// Mitsubishi GX Works2 project: finalfinal[1]   PLC: FX3G

// global labels: Global1
VAR_GLOBAL
  startDaySwitch AT X007 : BOOL;
  petelValue AT D1111 : REAL;
  petelTank AT D1101 : REAL;
  lemonValue AT D1114 : REAL;
  lemonTank AT D1103 : REAL;
  GummyBear AT D1118 : REAL;
  GummyBearTank AT D1120 : REAL;
  stabillizerValue AT D1106 : REAL;
  stabillizerTank AT D1127 : REAL;
  totalPackages AT D1108 : REAL;
  finished_timer AT TS5 : BOOL;
  GummyGumPackages AT D1108 : INT;
END_VAR
VAR_GLOBAL CONSTANT
  zeroPackages : REAL;
  amountOfPetelForOnePackage : REAL := 280;
  amountOfLemonForOnePackage : REAL := 455;
  amountOfStabillizerForOnePackage : REAL := 105;
  amountOfGummyBearForOnePackage : REAL := 28;
END_VAR
VAR_GLOBAL
  notEnoughForRegularGummyGam AT M23 : BOOL;
  notEnoughForPinukGummyGam AT M24 : BOOL;
END_VAR
VAR_GLOBAL CONSTANT
  amountOfPetelForPinukPack : REAL := 385;
  amountOfLemonForPinukPack : REAL := 665;
  amountOfStabillizerForPinukPack : REAL := 210;
  amountOfGummyBearForPinukPack : REAL := 70;
END_VAR
VAR_GLOBAL
  endDay AT M25 : BOOL;
  dayOn AT Y007 : BOOL;
  Sample AT X001 : BOOL;
  analogInput1 AT D8280 : INT;
  save AT D8000 : INT;
  saveAnalogInput AT D8000 : INT;
END_VAR
VAR_GLOBAL CONSTANT
  normalizeAnalog : REAL := 400;
END_VAR
VAR_GLOBAL
  gumygamType AT D1333 : REAL;
  chekType AT M116 : BOOL;
END_VAR
VAR_GLOBAL CONSTANT
  pinukThreshold : REAL := 5.0;
END_VAR
VAR_GLOBAL
  notEnoughMaterials AT M26 : BOOL;
  emergency AT X005 : BOOL;
END_VAR
VAR_GLOBAL CONSTANT
  amountOfPetel : REAL := 280;
  amountOfPetelP : REAL := 385;
  amountOfLemon : REAL := 665;
  amountOfLemonP : REAL := 665;
  amountOfStabillizerP : REAL := 210;
  amountOfPetelR : REAL := 280;
  amountOfLemonR : REAL := 455;
  amountOfStabillizerR : REAL := 105;
END_VAR
VAR_GLOBAL
  petelCream AT D1118 : REAL;
END_VAR
VAR_GLOBAL CONSTANT
  petelPinuk : REAL := 560;
  petelRegular : REAL := 350;
END_VAR
VAR_GLOBAL
  petelCreamP AT D1118 : REAL;
  lemonCreamP AT D1119 : REAL;
END_VAR
VAR_GLOBAL CONSTANT
  lemonPinuk : REAL := 700;
END_VAR
VAR_GLOBAL
  petelCreamR AT D1121 : REAL;
  lemonCreamR AT D1123 : REAL;
END_VAR
VAR_GLOBAL CONSTANT
  lemonRegular : REAL := 490;
END_VAR
VAR_GLOBAL
  StartIceCream AT M31 : BOOL;
  IceCreamTimer AT TC2 : BOOL;
END_VAR
VAR_GLOBAL CONSTANT
  readyIceCream : INT := 35;
END_VAR
VAR_GLOBAL
  IceCreamTimer1 AT TS2 : BOOL;
  temperatureBelow AT X005 : BOOL;
  Stiring AT Y000 : BOOL;
  striring AT Y000 : BOOL;
END_VAR
VAR_GLOBAL CONSTANT
  count5 : INT := 50;
END_VAR
VAR_GLOBAL
  startFreezing AT M124 : BOOL;
  startFreeze AT X002 : BOOL;
  endStageOne AT M122 : BOOL;
  petelIceCream AT D1118 : REAL;
  lemonIceCream AT D1139 : REAL;
  freezePetelIceCream AT D5555 : REAL;
  freezeLemonIceCream AT D6666 : REAL;
  finishFreeze AT M138 : BOOL;
  holdClock AT M128 : BOOL;
  startClock AT X007 : BOOL;
  mixingContainer AT D4444 : REAL;
END_VAR
VAR_GLOBAL CONSTANT
  amountOfGummtBearP : REAL := 70;
  amountOfGummtBearR : REAL := 28;
END_VAR
VAR_GLOBAL
  StartMix AT M140 : BOOL;
  notEnoughForPinuk AT M24 : BOOL;
  notEnoughForRegular AT M23 : BOOL;
  regularType AT M28 : BOOL;
END_VAR
VAR_GLOBAL CONSTANT
  freezeTime : INT := 80;
END_VAR
VAR_GLOBAL
  freezeTimer AT TC3 : BOOL;
  outFreeze AT TS3 : BOOL;
  freezeLight AT Y002 : BOOL;
  tempSwitch AT X003 : BOOL;
  freezeClockHolder AT M128 : BOOL;
  pinukType AT M29 : BOOL;
  timer0 AT TC0 : BOOL;
END_VAR
VAR_GLOBAL CONSTANT
  timepinuk : REAL := 50;
  timregular : REAL := 30;
END_VAR
VAR_GLOBAL
  timeForMix AT D7775 : REAL;
  outTimer0 AT TS0 : BOOL;
  finished_Mixing AT M53 : BOOL;
  outTimer2 AT TS5 : BOOL;
  startFlashing AT M0 : BOOL;
  Switch1 AT Y005 : BOOL;
  timer1 AT TC4 : BOOL;
END_VAR
VAR_GLOBAL CONSTANT
  count1 : INT := 10;
END_VAR
VAR_GLOBAL
  outTimer1 AT TS4 : BOOL;
  Switch2 AT Y006 : BOOL;
  timer2 AT TC5 : BOOL;
  StartPacking AT X004 : BOOL;
  packOneGummyGam AT X000 : BOOL;
  countOne AT CC1 : BOOL;
END_VAR
VAR_GLOBAL CONSTANT
  oneGummyGam : INT := 1;
END_VAR
VAR_GLOBAL
  endOne AT CS1 : BOOL;
  endPack AT CS2 : BOOL;
  SwitchOneGummy AT Y004 : BOOL;
END_VAR
VAR_GLOBAL CONSTANT
  normalizeAnalog1 : REAL := 400;
END_VAR
VAR_GLOBAL
  timer_1 AT TC4 : BOOL;
  outTimer_1 AT TS4 : BOOL;
  finished_timer_freeze AT M61 : BOOL;
  canStartFreeze AT M120 : BOOL;
  StartIceCream1 : BOOL;
END_VAR
VAR_GLOBAL CONSTANT
  zero : REAL;
END_VAR
VAR_GLOBAL
  letsFlash AT M72 : BOOL;
  countPack AT CC2 : BOOL;
END_VAR
VAR_GLOBAL CONSTANT
  SixMoreGummyGam : WORD := 7;
END_VAR
VAR_GLOBAL
  finishPack AT CS2 : BOOL;
END_VAR
VAR_GLOBAL CONSTANT
  more7 : REAL := 7;
  morePack : REAL := 1;
  sevenMore : INT := 7;
END_VAR
VAR_GLOBAL
  output_analog AT D8282 : INT;
  restart AT M100 : BOOL;
END_VAR

// task Task_01 (event TRUE, interval 0, priority 31): POU_01

PROGRAM POU_01
(* structured ladder/FBD written out as ST: instructions are called as NAME(EN, inputs, outputs); _pN, _eN, _tN stand for wires *)
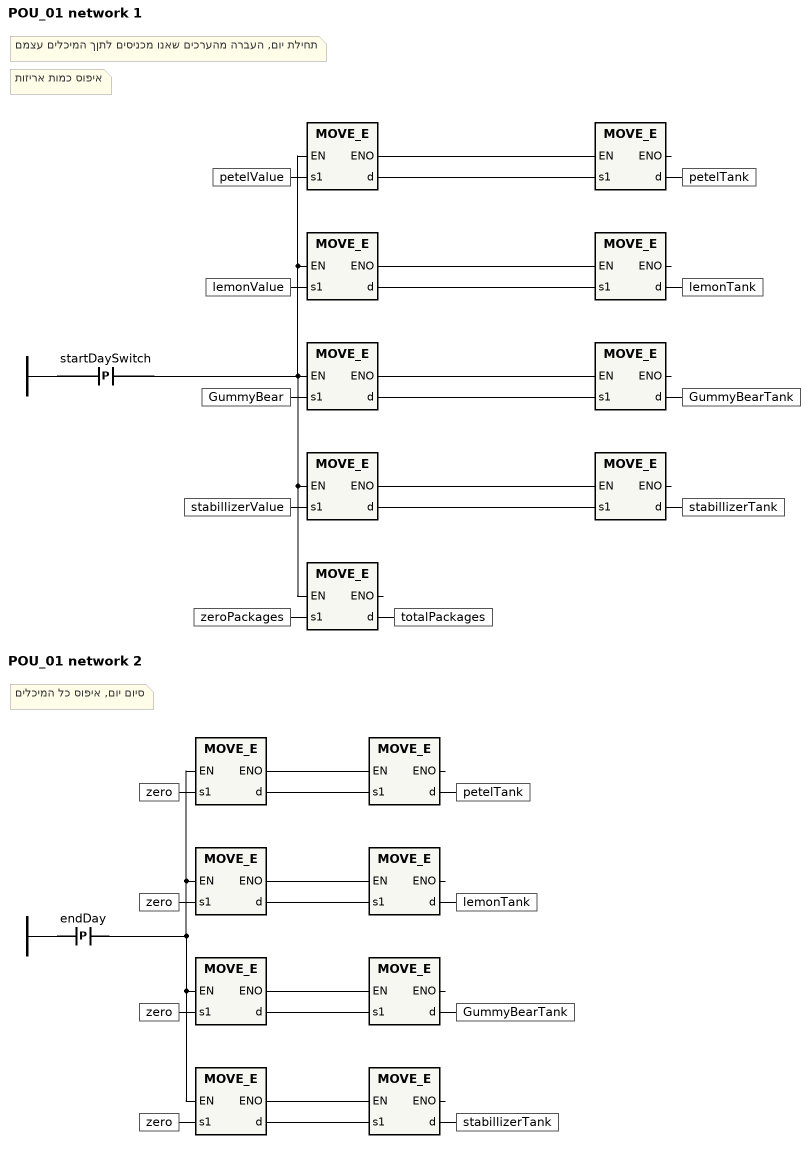
(* network 1 *)
(* תחילת יום, העברה מהערכים שאנו מכניסים לתןך המיכלים עצמם *)
(* איפוס כמות אריזות *)
_p1 := LDP(TRUE, startDaySwitch);
_e3 := MOVE_E(_p1, petelValue, _t2);
MOVE_E(_e3, _t2, petelTank);
_e5 := MOVE_E(_p1, lemonValue, _t4);
MOVE_E(_e5, _t4, lemonTank);
_e7 := MOVE_E(_p1, GummyBear, _t6);
MOVE_E(_e7, _t6, GummyBearTank);
_e9 := MOVE_E(_p1, stabillizerValue, _t8);
MOVE_E(_e9, _t8, stabillizerTank);
MOVE_E(_p1, zeroPackages, totalPackages);
(* network 2 *)
(* סיום יום, איפוס כל המיכלים *)
_p1 := LDP(TRUE, endDay);
_e3 := MOVE_E(_p1, zero, _t2);
MOVE_E(_e3, _t2, petelTank);
_e5 := MOVE_E(_p1, zero, _t4);
MOVE_E(_e5, _t4, lemonTank);
_e7 := MOVE_E(_p1, zero, _t6);
MOVE_E(_e7, _t6, GummyBearTank);
_e9 := MOVE_E(_p1, zero, _t8);
MOVE_E(_e9, _t8, stabillizerTank);
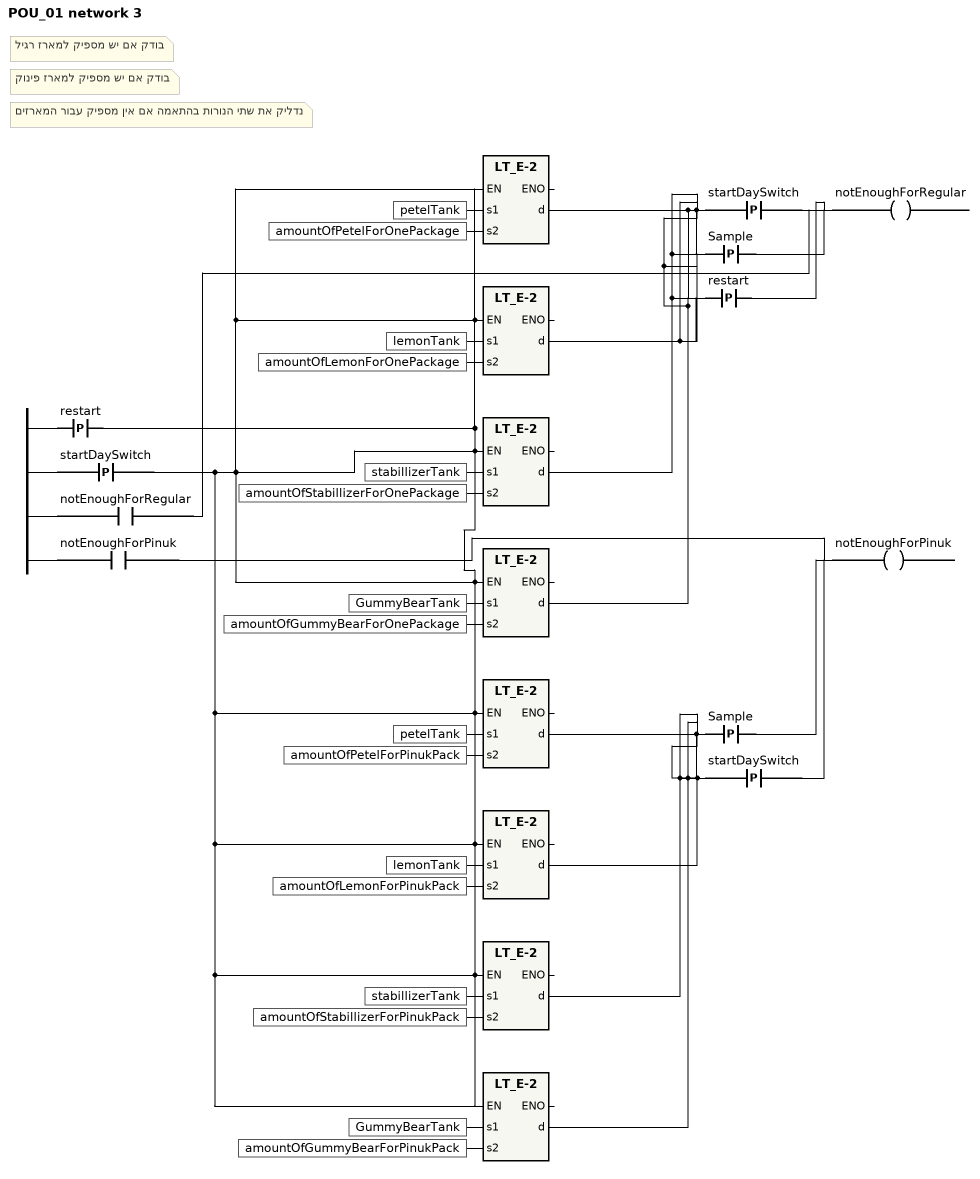
(* network 3 *)
(* בודק אם יש מספיק למארז רגיל *)
(* בודק אם יש מספיק למארז פינוק *)
(* נדליק את שתי הנורות בהתאמה אם אין מספיק עבור המארזים *)
_p1 := LDP(TRUE, restart) OR LDP(TRUE, startDaySwitch);
LT_E(_p1, petelTank, amountOfPetelForOnePackage, _t2);
LT_E(_p1, lemonTank, amountOfLemonForOnePackage, _t3);
LT_E(_p1, stabillizerTank, amountOfStabillizerForOnePackage, _t4);
LT_E(_p1, GummyBearTank, amountOfGummyBearForOnePackage, _t5);
_p6 := _t2 OR _t3 OR _t4 OR _t5;
notEnoughForRegular := (_p6 AND LDP(TRUE, startDaySwitch)) OR (_p6 AND LDP(TRUE, Sample)) OR (_p6 AND LDP(TRUE, restart)) OR notEnoughForRegular;
LT_E(_p1, petelTank, amountOfPetelForPinukPack, _t7);
LT_E(_p1, lemonTank, amountOfLemonForPinukPack, _t8);
LT_E(_p1, stabillizerTank, amountOfStabillizerForPinukPack, _t9);
LT_E(_p1, GummyBearTank, amountOfGummyBearForPinukPack, _t10);
_p11 := _t7 OR _t8 OR _t9 OR _t10;
notEnoughForPinuk := (_p11 AND LDP(TRUE, Sample)) OR (_p11 AND LDP(TRUE, startDaySwitch)) OR notEnoughForPinuk;
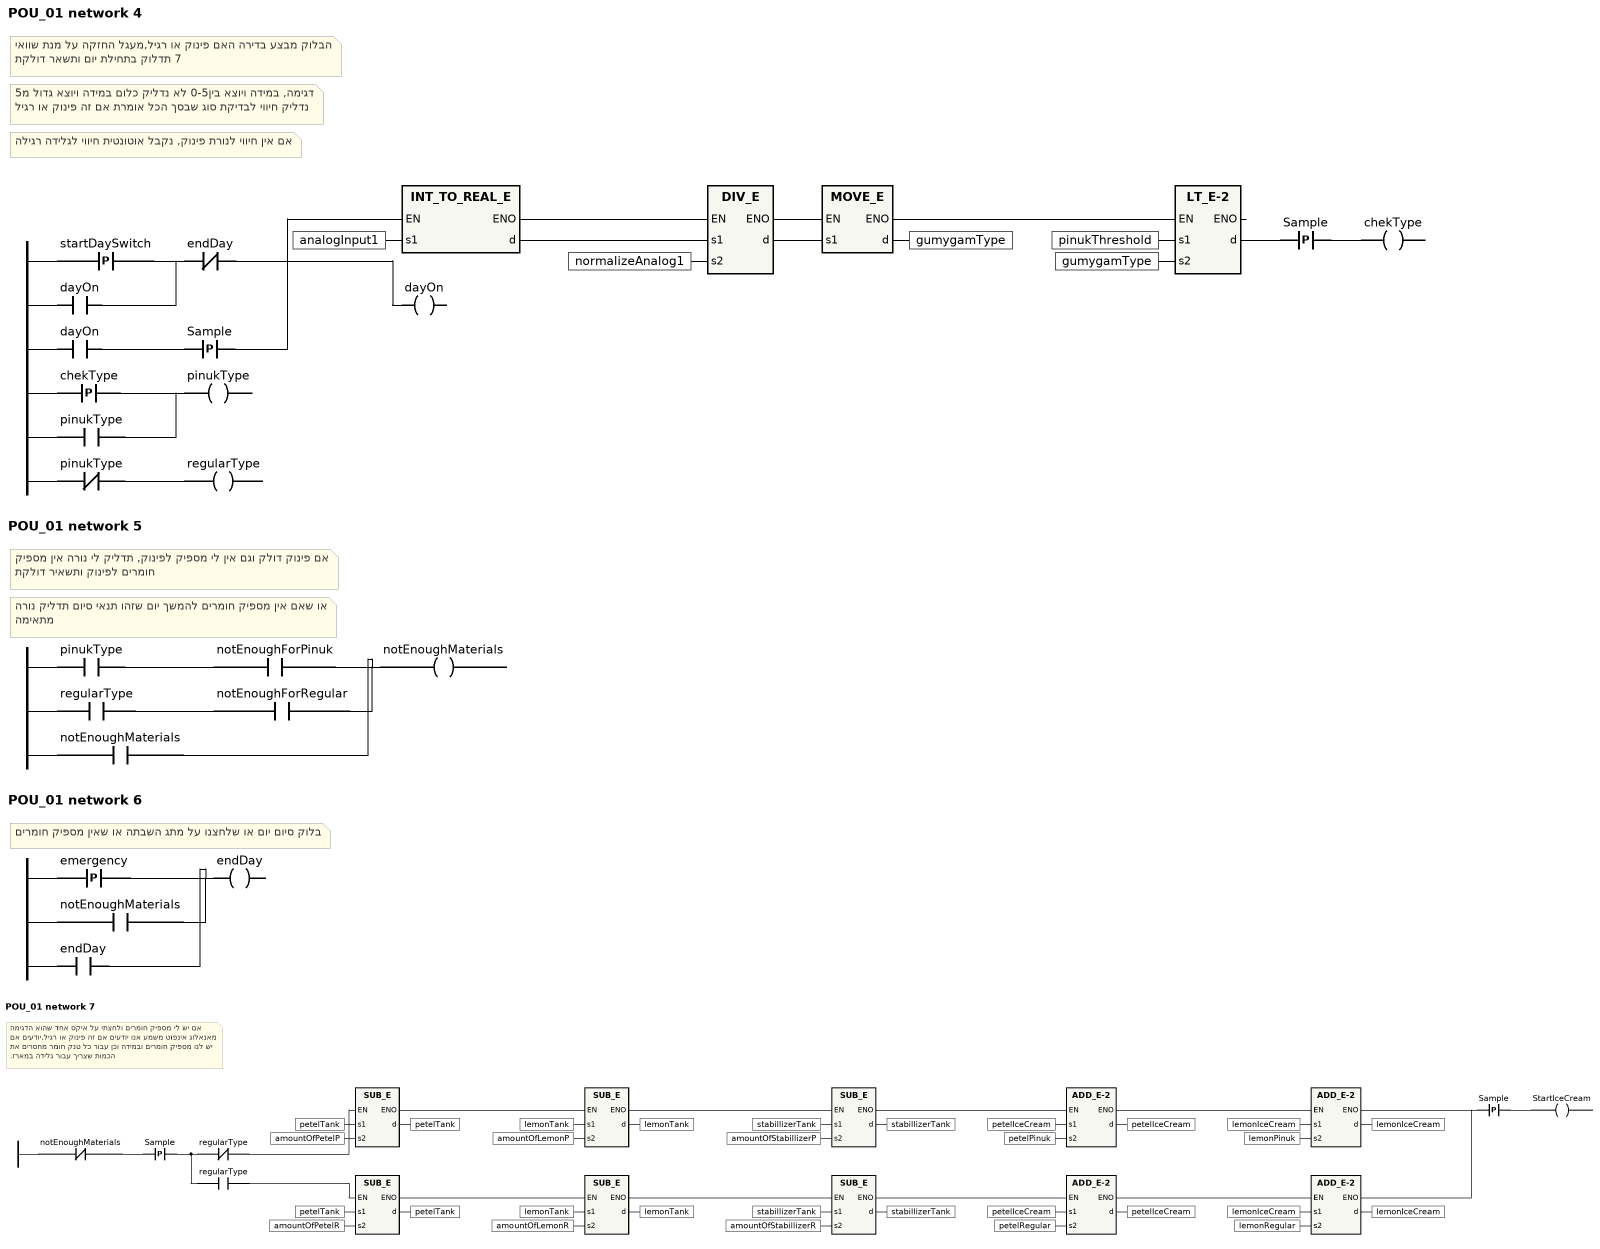
(* network 4 *)
(* הבלוק מבצע בדירה האם פינוק או רגיל,מעגל החזקה על מנת שוואי 7 תדלוק בתחילת יום ותשאר דולקת *)
(* דגימה, במידה ויוצא בין0-5 לא נדליק כלום במידה ויוצא גדול מ5 נדליק חיווי לבדיקת סוג שבסך הכל אומרת אם זה פינוק או רגיל *)
(* אם אין חיווי לנורת פינוק, נקבל אוטונטית חיווי לגלידה רגילה *)
dayOn := (LDP(TRUE, startDaySwitch) OR dayOn) AND NOT endDay;
_e2 := INT_TO_REAL_E(dayOn AND LDP(TRUE, Sample), analogInput1, _t1);
_e4 := DIV_E(_e2, _t1, normalizeAnalog1, _t3);
_e5 := MOVE_E(_e4, _t3, gumygamType);
LT_E(_e5, pinukThreshold, gumygamType, _t6);
chekType := _t6 AND LDP(TRUE, Sample);
pinukType := LDP(TRUE, chekType) OR pinukType;
regularType := NOT pinukType;
(* network 5 *)
(* אם פינוק דולק וגם אין לי מספיק לפינוק, תדליק לי נורה אין מספיק חומרים לפינוק ותשאיר דולקת *)
(* או שאם אין מספיק חומרים להמשך יום שזהו תנאי סיום תדליק נורה מתאימה *)
notEnoughMaterials := (pinukType AND notEnoughForPinuk) OR (regularType AND notEnoughForRegular) OR notEnoughMaterials;
(* network 6 *)
(* בלוק סיום יום או שלחצנו על מתג השבתה או שאין מספיק חומרים *)
endDay := LDP(TRUE, emergency) OR notEnoughMaterials OR endDay;
(* network 7 *)
(* אם יש לי מספיק חומרים ולחצתי על איקס אחד שהוא הדגימה מאנאלוג אינפוט משמע אנו יודעים אם זה פינוק או רגיל,יודעים אם יש לנו מספיק חומרים ובמידה וכן עבור כל טנק חומר מחסרים את הכמות שצריך עבור גלידה במארז. *)
_p1 := NOT notEnoughMaterials AND LDP(TRUE, Sample);
_e2 := SUB_E(_p1 AND NOT regularType, petelTank, amountOfPetelP, petelTank);
_e3 := SUB_E(_e2, lemonTank, amountOfLemonP, lemonTank);
_e4 := SUB_E(_e3, stabillizerTank, amountOfStabillizerP, stabillizerTank);
_e5 := ADD_E(_e4, petelIceCream, petelPinuk, petelIceCream);
_e6 := ADD_E(_e5, lemonIceCream, lemonPinuk, lemonIceCream);
_e7 := SUB_E(_p1 AND regularType, petelTank, amountOfPetelR, petelTank);
_e8 := SUB_E(_e7, lemonTank, amountOfLemonR, lemonTank);
_e9 := SUB_E(_e8, stabillizerTank, amountOfStabillizerR, stabillizerTank);
_e10 := ADD_E(_e9, petelIceCream, petelRegular, petelIceCream);
_e11 := ADD_E(_e10, lemonIceCream, lemonRegular, lemonIceCream);
StartIceCream := (_e6 OR _e11) AND LDP(TRUE, Sample);
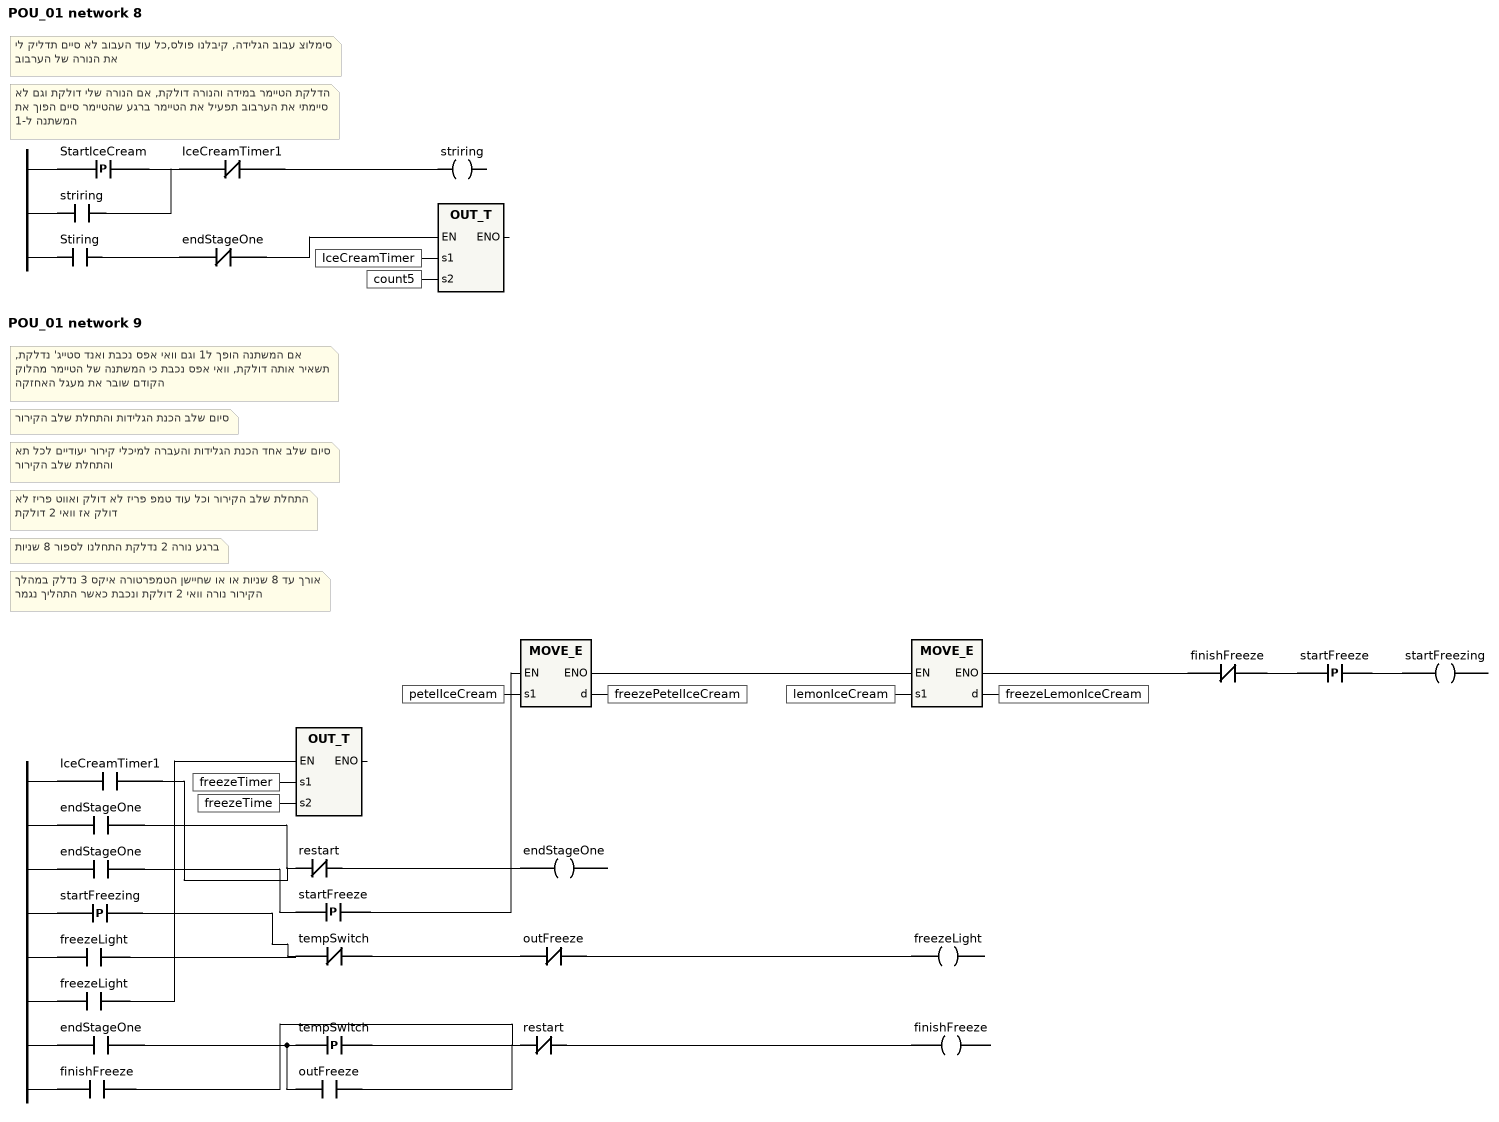
(* network 8 *)
(* סימלוצ עבוב הגלידה, קיבלנו פולס,כל עוד העבוב לא סיים תדליק לי את הנורה של הערבוב *)
(* הדלקת הטיימר במידה והנורה דולקת, אם הנורה שלי דולקת וגם לא סיימתי את הערבוב תפעיל את הטיימר ברגע שהטיימר סיים הפוך את המשתנה ל-1 *)
striring := (LDP(TRUE, StartIceCream) OR striring) AND NOT IceCreamTimer1;
OUT_T(Stiring AND NOT endStageOne, IceCreamTimer, count5);
(* network 9 *)
(* אם המשתנה הופך ל1 וגם וואי אפס נכבת ואנד סטייג' נדלקת, תשאיר אותה דולקת, וואי אפס נכבת כי המשתנה של הטיימר מהלוק הקודם שובר את מעגל האחזקה *)
(* סיום שלב הכנת הגלידות והתחלת שלב הקירור *)
(* סיום שלב אחד הכנת הגלידות והעברה למיכלי קירור יעודיים לכל תא והתחלת שלב הקירור *)
(* התחלת שלב הקירור וכל עוד טמפ פריז לא דולק ואווט פריז לא דולק אז וואי 2 דולקת *)
(* ברגע נורה 2 נדלקת התחלנו לספור 8 שניות *)
(* אורך עד 8 שניות או או שחיישן הטמפרטורה איקס 3 נדלק במהלך הקירור נורה וואי 2 דולקת ונכבת כאשר התהליך נגמר *)
endStageOne := (IceCreamTimer1 OR endStageOne) AND NOT restart;
_e1 := MOVE_E(endStageOne AND LDP(TRUE, startFreeze), petelIceCream, freezePetelIceCream);
_e2 := MOVE_E(_e1, lemonIceCream, freezeLemonIceCream);
startFreezing := _e2 AND NOT finishFreeze AND LDP(TRUE, startFreeze);
freezeLight := ((LDP(TRUE, startFreezing) OR freezeLight) AND NOT tempSwitch) AND NOT outFreeze;
OUT_T(freezeLight, freezeTimer, freezeTime);
finishFreeze := ((endStageOne AND LDP(TRUE, tempSwitch)) OR (endStageOne AND outFreeze) OR finishFreeze) AND NOT restart;
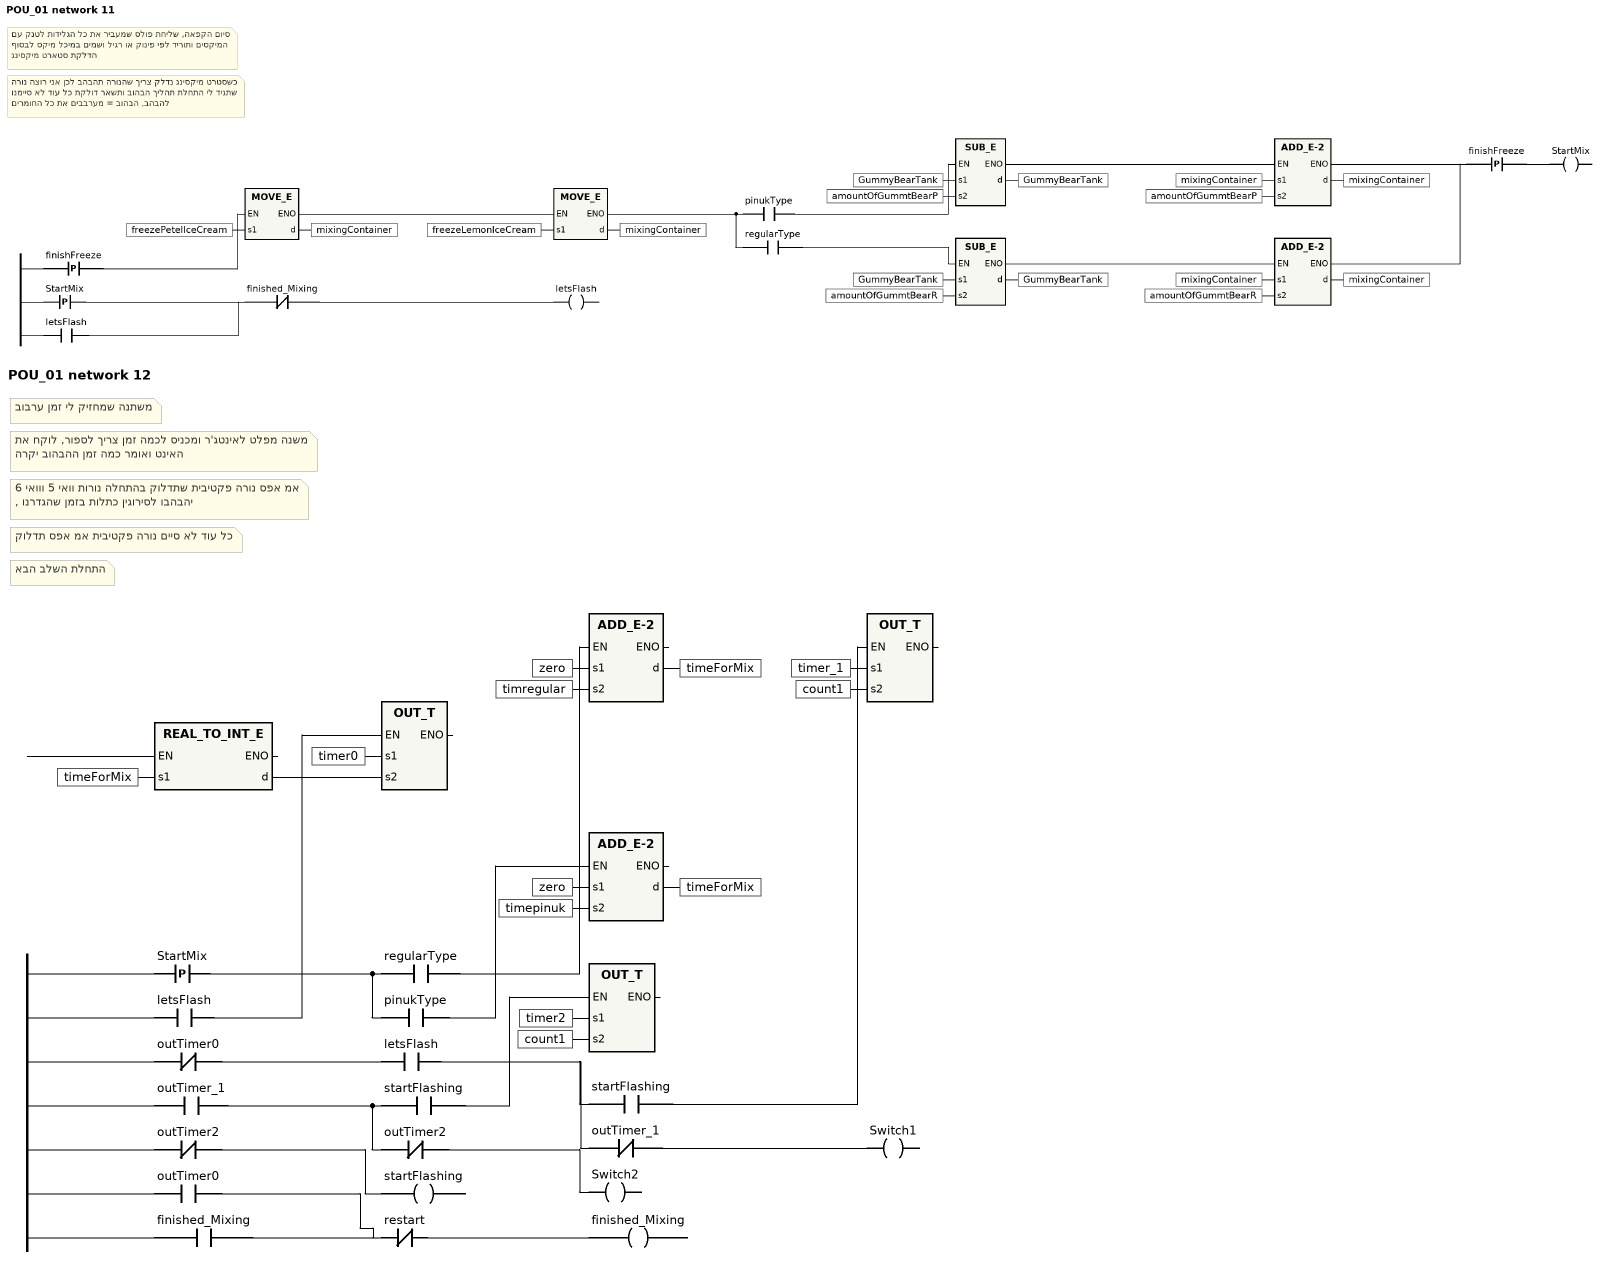
(* network 11 *)
(* סיום הקפאה, שליחת פולס שמעביר את כל הגלידות לטנק עם המיקסים ותוריד לפי פינוק או רגיל ושמים במיכל מיקס לבסוף הדלקת סטארט מיקסינג *)
(* כשסטרט מיקסינג נדלק צריך שהנורה תהבהב לכן אני רוצה נורה שתגיד לי התחלת תהליך הבהוב ותשאר דולקת כל עוד לא סיימנו להבהב, הבהוב = מערבבים את כל החומרים *)
_e1 := MOVE_E(LDP(TRUE, finishFreeze), freezePetelIceCream, mixingContainer);
_e2 := MOVE_E(_e1, freezeLemonIceCream, mixingContainer);
_e3 := SUB_E(_e2 AND pinukType, GummyBearTank, amountOfGummtBearP, GummyBearTank);
_e4 := ADD_E(_e3, mixingContainer, amountOfGummtBearP, mixingContainer);
_e5 := SUB_E(_e2 AND regularType, GummyBearTank, amountOfGummtBearR, GummyBearTank);
_e6 := ADD_E(_e5, mixingContainer, amountOfGummtBearR, mixingContainer);
StartMix := (_e4 OR _e6) AND LDP(TRUE, finishFreeze);
letsFlash := (LDP(TRUE, StartMix) OR letsFlash) AND NOT finished_Mixing;
(* network 12 *)
(* משתנה שמחזיק לי זמן ערבוב *)
(* משנה מפלט לאינטג'ר ומכניס לכמה זמן צריך לספור, לוקח את האינט ואומר כמה זמן ההבהוב יקרה *)
(* אמ אפס נורה פקטיבית שתדלוק בהתחלה נורות וואי 5 ווואי 6 יהבהבו לסירוגין כתלות בזמן שהגדרנו , *)
(* כל עוד לא סיים נורה פקטיבית אמ אפס תדלוק *)
(* התחלת השלב הבא *)
_p1 := LDP(TRUE, StartMix);
ADD_E(_p1 AND regularType, zero, timregular, timeForMix);
ADD_E(_p1 AND pinukType, zero, timepinuk, timeForMix);
REAL_TO_INT_E(TRUE, timeForMix, _t2);
OUT_T(letsFlash, timer0, _t2);
_p3 := NOT outTimer0 AND letsFlash;
OUT_T(_p3 AND startFlashing, timer_1, count1);
Switch1 := _p3 AND NOT outTimer_1;
OUT_T(outTimer_1 AND startFlashing, timer2, count1);
Switch2 := outTimer_1 AND NOT outTimer2;
startFlashing := NOT outTimer2;
finished_Mixing := (outTimer0 OR finished_Mixing) AND NOT restart;
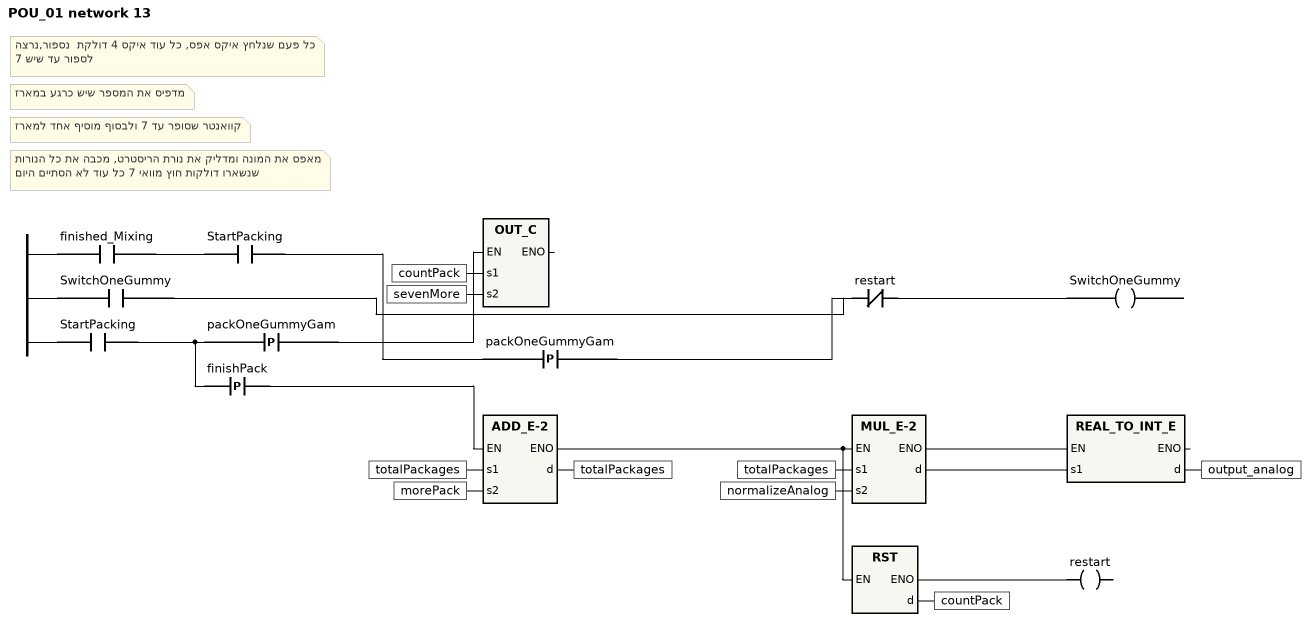
(* network 13 *)
(* כל פעם שנלחץ איקס אפס, כל עוד איקס 4 דולקת  נספור,נרצה לספור עד שיש 7 *)
(* מדפיס את המספר שיש כרגע במארז *)
(* קוואנטר שסופר עד 7 ולבסוף מוסיף אחד למארז *)
(* מאפס את המונה ומדליק את נורת הריסטרט, מכבה את כל הנורות שנשארו דולקות חוץ מוואי 7 כל עוד לא הסתיים היום *)
SwitchOneGummy := ((finished_Mixing AND StartPacking AND LDP(TRUE, packOneGummyGam)) OR SwitchOneGummy) AND NOT restart;
_e1 := ADD_E(StartPacking AND LDP(TRUE, finishPack), totalPackages, morePack, totalPackages);
_e3 := MUL_E(_e1, totalPackages, normalizeAnalog, _t2);
REAL_TO_INT_E(_e3, _t2, output_analog);
OUT_C(StartPacking AND LDP(TRUE, packOneGummyGam), countPack, sevenMore);
_e4 := RST(_e1, countPack);
restart := _e4;
END_PROGRAM
